TYPE U_OdriveSetControllerModeBytes :
UNION
    stSetControllerMode : ST_OdriveSetControllerMode;
    aBytes : ARRAY[0..7] OF BYTE;
END_UNION
END_TYPE

(* stored: Version 1.1.0.1
   DUT U_OdriveSetControllerModeBytes: Id {c3556745-197d-4417-abd2-c255c4c95511} *)
